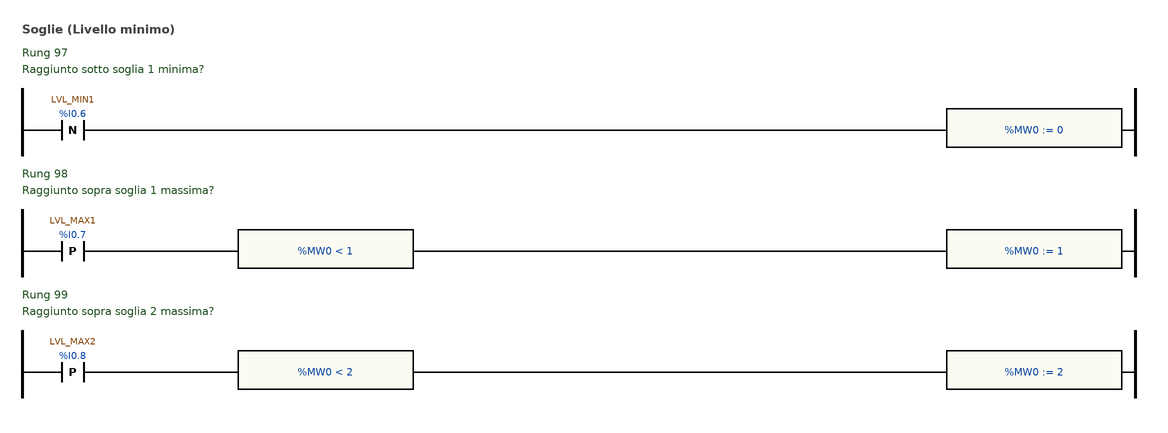
[picture p24: Soglie (Livello minimo), ladder]

// Rung 97
// Raggiunto sotto soglia 1 minima?
  LDF %I0.6               (* LVL_MIN1 *)
  [ %MW0 := 0 ]           (* NUM_POMPE_DA_COMANDARE *)
  // as ST:
  //   IF FALLING(LVL_MIN1) THEN NUM_POMPE_DA_COMANDARE := 0; END_IF;

// Rung 98
// Raggiunto sopra soglia 1 massima?
  LDR %I0.7               (* LVL_MAX1 *)
  AND [ %MW0 < 1 ]        (* NUM_POMPE_DA_COMANDARE *)
  [ %MW0 := 1 ]           (* NUM_POMPE_DA_COMANDARE *)
  // as ST:
  //   IF RISING(LVL_MAX1) AND NUM_POMPE_DA_COMANDARE < 1 THEN NUM_POMPE_DA_COMANDARE := 1; END_IF;

// Rung 99
// Raggiunto sopra soglia 2 massima?
  LDR %I0.8               (* LVL_MAX2 *)
  AND [ %MW0 < 2 ]        (* NUM_POMPE_DA_COMANDARE *)
  [ %MW0 := 2 ]           (* NUM_POMPE_DA_COMANDARE *)
  // as ST:
  //   IF RISING(LVL_MAX2) AND NUM_POMPE_DA_COMANDARE < 2 THEN NUM_POMPE_DA_COMANDARE := 2; END_IF;
